# EPICS substitutions: iocBoot/ioc13lab/Pelco_CM6700.substitutions
file "$(IP)/db/Pelco_CM6700.db"
{
pattern
{P,       R,       PORT}
{13LAB:,  Pelco1,  serial5}
}

file "$(IP)/db/Pelco_CM6700_names.db"
{
pattern
{P,       R,       STR}
{13LAB:,  Pelco1,  ZRST}
{13LAB:,  Pelco1,  ONST}
{13LAB:,  Pelco1,  TWST}
{13LAB:,  Pelco1,  THST}
{13LAB:,  Pelco1,  FRST}
{13LAB:,  Pelco1,  FVST}
{13LAB:,  Pelco1,  SXST}
{13LAB:,  Pelco1,  SVST}
{13LAB:,  Pelco1,  EIST}
{13LAB:,  Pelco1,  NIST}
{13LAB:,  Pelco1,  TEST}
{13LAB:,  Pelco1,  ELST}
{13LAB:,  Pelco1,  TVST}
{13LAB:,  Pelco1,  TTST}
{13LAB:,  Pelco1,  FTST}
{13LAB:,  Pelco1,  FFST}
}
